// TIA Portal V19 export
TYPE "TExtEncoder_Alarms"
// stored: Access Published
   STRUCT
      TOEncoder : Bool;   // Alarm in technology object
      MCFunction : Bool;   // Alarm of MC function
      TimeOutExecution : Bool;   // Time out power on encoder
   END_STRUCT;
END_TYPE
